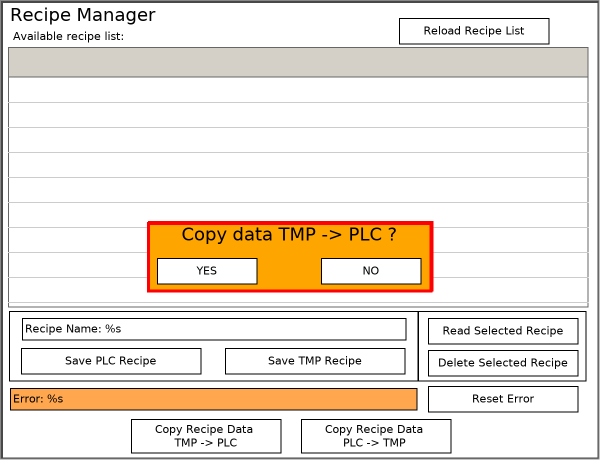
VISUALIZATION vRecManDialog  // 600x460
VAR_IN_OUT
	fbRecipe:fbRecMan;
END_VAR
    Rectangle (1,1 598x458)
    Rectangle (418,311 168x70)
    Rectangle (9,311 409x70)
    Table (8,47 580x260), data array: fbRecipe.astRecipeList
        p1128707560: fbRecipe.iNbOfFoundRecipes
        p1137915858: fbRecipe.iTableSelIndex
        p1822360349: fbRecipe.bTableRowSelected
        p3854506369: fbRecipe.astRecipeList[INDEX].sFileName
        p1892666644: fbRecipe.astRecipeList[INDEX].dtCreationTime
        p2232123230: Recipe Name
        p511219082: Creation Time
    Label (7,0 150x30), "Recipe Manager"
    Label (10,29 150x15), "Available recipe list:"
    RoundedRectangle (399,18 150x26), "Reload Recipe List", colour toggle: fbRecipe.bRefreshingRecipeList
        toggle fbRecipe.bReloadRecipes
    RoundedRectangle (21,348 180x26), "Save PLC Recipe", colour toggle: fbRecipe.bWritingRecipe
        OnMouseClick: execute { fbRecipe.bWriteRecipe := NOT fbRecipe.bWriteRecipe; fbRecipe.bSavePLCStruct := TRUE; }
    Rectangle (22,318 384x22), "Recipe Name: %s", text variable: fbRecipe.sRecipeName
        OnMouseClick: write fbRecipe.sRecipeName via Default, title 'New Recipe Name', format %s
    RoundedRectangle (131,419 150x34), "Copy Recipe Data TMP -> PLC", colour toggle: fbRecipe.bCopyTMP_2_PLC
        toggle fbRecipe.bCopyTMP_2_PLC
    RoundedRectangle (301,419 150x34), "Copy Recipe Data PLC -> TMP", colour toggle: fbRecipe.bCopyPLC_2_TMP
        toggle fbRecipe.bCopyPLC_2_TMP
    RoundedRectangle (428,318 150x26), "Read Selected Recipe", colour toggle: fbRecipe.bReadingRecipe
        toggle fbRecipe.bReadRecipe
    RoundedRectangle (225,348 180x26), "Save TMP Recipe", colour toggle: fbRecipe.bWritingRecipe
        OnMouseClick: execute { fbRecipe.bWriteRecipe := NOT fbRecipe.bWriteRecipe; fbRecipe.bSavePLCStruct := FALSE; }
    Rectangle (10,388 407x22), "Error: %s", text variable: fbRecipe.nErrorCode, invisible if: NOT fbRecipe.bError
        OnMouseClick: write fbRecipe.sRecipeName via Default, title 'New Recipe Name', format %s
    RoundedRectangle (428,386 150x26), "Reset Error", colour toggle: fbRecipe.bResetInternal, invisible if: NOT fbRecipe.bError
        toggle fbRecipe.bResetInternal
    RoundedRectangle (428,350 150x26), "Delete Selected Recipe", colour toggle: fbRecipe.bDeletingRecipe
        toggle fbRecipe.bDeleteRecipe
    Group (148,221 285x70), invisible if: NOT fbRecipe.bDeleteRecipe
        Rectangle (0,0 285x70), "Delete selection ?"
        RoundedRectangle (10,36 100x26), "YES"
            toggle fbRecipe.bDeleteConfirmed
        RoundedRectangle (174,36 100x26), "NO"
            toggle fbRecipe.bDeleteRecipe
    Group (147,222 285x70), invisible if: NOT fbRecipe.bCopyTMP_2_PLC
        Rectangle (0,0 285x70), "Copy data TMP -> PLC ?"
        RoundedRectangle (10,36 100x26), "YES"
            toggle fbRecipe.bCopyTMP_2_PLC_Confirmed
        RoundedRectangle (174,36 100x26), "NO"
            toggle fbRecipe.bCopyTMP_2_PLC
END_VISUALIZATION

(* stored: Version 1.1.0.1, ProductVersion 3.1.4024.12
   Visu vRecManDialog: Id {83134544-57bb-4bd0-8471-f616b6f11adf} *)
